(* NC axis ctrl for EL7201 via EtherCAT *)
FUNCTION_BLOCK FB_MC2_EL7201AxisCtrl
VAR_INPUT
	bEnable				: BOOL;		(* set TRUE to enable axis and drive *)
	bReset				: BOOL;		(* set TRUE to reset axis or drive from ERROR condition *)
	bEnableRevDir		: BOOL;		(* set TRUE to allow axis to run in reverse direction *)
	fOverride			: LREAL;	(* max axis output in % *)
	bFastStop			: BOOL;		(* set TRUE to override RUN signals and stop axis immediately *)
	bRunVelo			: BOOL;		(* set TRUE to run axis at specified velocity, set FALSE to stop at specified pos *)
	bStopAtPos			: BOOL;		(* set TRUE to run axis at specified velocity, set FALSE to stop at specified pos *)
	bJogFwd				: BOOL;		(* set TRUE to jog forwards *)
	bJogRev				: BOOL;		(* set TRUE to jog reverse *)
	fStopPos			: LREAL;	(* target stop position *)
	fSetVelo			: LREAL;	(* target velocity *)
	fJogVelo			: LREAL;	(* jog velocity (does not take effect if jog is in progress *)
	sRamps				: ST_AxisCtrlRamps;	(* ramps for FastStop, Normal and Jog *)
	nEtherCATState		: UINT;		(* EtherCAT operating state *)
END_VAR
VAR_IN_OUT
	sParamSet			: ST_AxisParameterSet;	(* axis parameter set *)
	sAxis				: AXIS_REF;	(* NC axis structure *)
END_VAR
VAR_OUTPUT
	bInitOK				: BOOL;		(* TRUE = parameter set read at least once *)
	bEnabled			: BOOL;		(* TRUE = axis is enabled *)
	bActive				: BOOL;		(* TRUE = axis is moving *)
	bJogActive			: BOOL;		(* TRUE = axis is moving in JOG mode *)
	bRunningFwd			: BOOL;		(* TRUE = axis is running forwards *)
	bRunningRev			: BOOL;		(* TRUE = axis is running backwards *)
	bHomed				: BOOL;		(* TRUE = axis has been homed *)
	bAxisError			: BOOL;		(* TRUE = axis is in error state *)
	nAxisErrorID		: UDINT;	(* NC axis error code *)

	fActPos				: LREAL;	(* axis absolute position *)
	fModuloPos			: LREAL;	(* axis modulo position *)
	fActVelo			: LREAL;	(* axis actual velocity *)
	bDriveError			: BOOL;		(* TRUE = EL7201 error active *)
	nStatusDWord		: DWORD;		(* drive status code *)
	fAmplifierTemp		: LREAL;	(* Amplifier temperature (degrees) *)
	fDCLinkVolts		: LREAL;	(* DC link voltage (volts) *)
END_VAR
VAR
	fbAxisCtrl			: FB_MC2_BasicAxisCtrl;
	fbEtherCATDelay		: TON;
	fbVeloCtrl			: FB_MC2_VeloCtrl;
	fbDriveReset		: MC_Reset;
	fbDriveAddr			: MC_ReadDriveAddress;
	fbDriveStatus		: FB_MC2_EL7201Status;
END_VAR
(*
-------------------------------------------------------------------------------------------------
Date		Version	Author	Comments
-------------------------------------------------------------------------------------------------
30/01/2015	3.00.00	PB		Updated with new FB_MC2_BasicAxisCtrl.
							MC_Reset for DriveReset now phased with fbSyncTimer in FB_MC2_BasicAxisCtrl.
							EL7201 status info (Warning, AmplifierTemp and DCLinkVolts) read via EtherCAT acyclic channel .
							
-------------------------------------------------------------------------------------------------
17/10/2012	1.09.02	PB		MC_Reset added to clear DriveError. as this does not cause Axis Error.
							FB_MC2_BasicAxisCtrl only issues reset if AxisError is active but DriveError on EL7201 does not cause AxisError.
21/12/2011	1.08.00	PB		Initial release

-------------------------------------------------------------------------------------------------
*)
VAR // added by the converter: edge detectors and wires of the graphical bodies
    _w1 : BOOL;
END_VAR

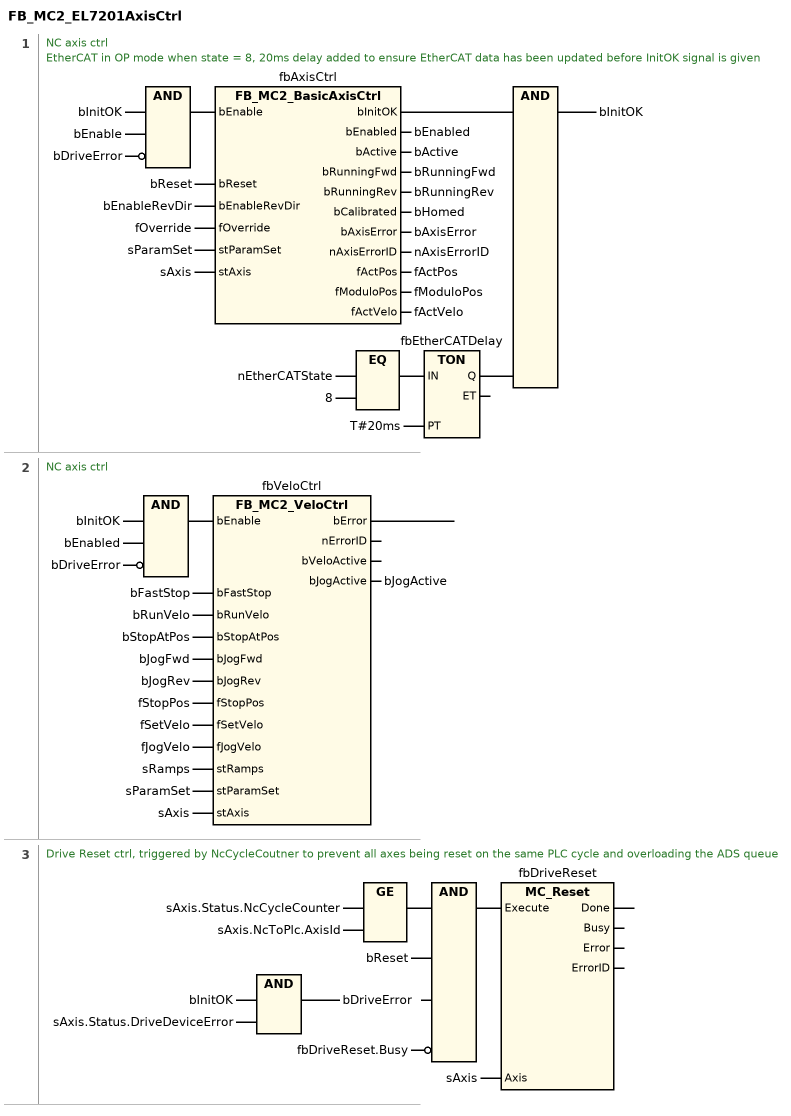
// NETWORK 1
// 					NC axis ctrl
// EtherCAT in OP mode when state = 8, 20ms delay added to ensure EtherCAT data has been updated before InitOK signal is given
//
fbAxisCtrl(
    bEnable := bInitOK AND bEnable AND NOT bDriveError,
    bReset := bReset,
    bEnableRevDir := bEnableRevDir,
    fOverride := fOverride,
    stParamSet := sParamSet,
    stAxis := sAxis,
    bEnabled => bEnabled,
    bActive => bActive,
    bRunningFwd => bRunningFwd,
    bRunningRev => bRunningRev,
    bCalibrated => bHomed,
    bAxisError => bAxisError,
    nAxisErrorID => nAxisErrorID,
    fActPos => fActPos,
    fModuloPos => fModuloPos,
    fActVelo => fActVelo); // FB_MC2_BasicAxisCtrl
fbEtherCATDelay(IN := nEtherCATState = 8, PT := T#20ms); // TON
bInitOK := fbAxisCtrl.bInitOK AND fbEtherCATDelay.Q;

// NETWORK 2
// NC axis ctrl
fbVeloCtrl(
    bEnable := bInitOK AND bEnabled AND NOT bDriveError,
    bFastStop := bFastStop,
    bRunVelo := bRunVelo,
    bStopAtPos := bStopAtPos,
    bJogFwd := bJogFwd,
    bJogRev := bJogRev,
    fStopPos := fStopPos,
    fSetVelo := fSetVelo,
    fJogVelo := fJogVelo,
    stRamps := sRamps,
    stParamSet := sParamSet,
    stAxis := sAxis,
    bJogActive => bJogActive); // FB_MC2_VeloCtrl

// NETWORK 3
// Drive Reset ctrl, triggered by NcCycleCoutner to prevent all axes being reset on the same PLC cycle and overloading the ADS queue
_w1 := bInitOK AND sAxis.Status.DriveDeviceError;
bDriveError := _w1;
fbDriveReset(Execute := sAxis.Status.NcCycleCounter >= sAxis.NcToPlc.AxisId AND bReset AND _w1 AND NOT fbDriveReset.Busy, Axis := sAxis); // MC_Reset

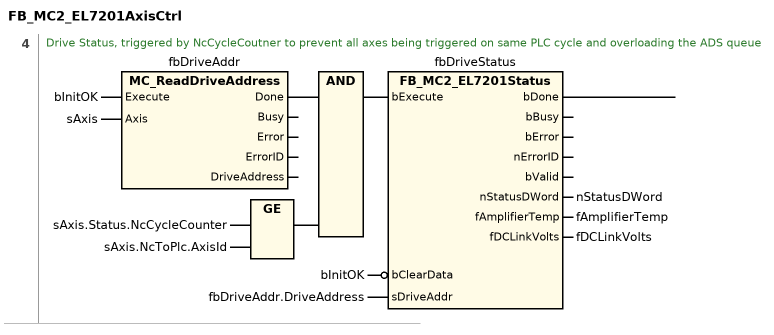
// NETWORK 4
// Drive Status, triggered by NcCycleCoutner to prevent all axes being triggered on same PLC cycle and overloading the ADS queue
fbDriveAddr(Execute := bInitOK, Axis := sAxis); // MC_ReadDriveAddress
fbDriveStatus(
    bExecute := fbDriveAddr.Done AND sAxis.Status.NcCycleCounter >= sAxis.NcToPlc.AxisId,
    bClearData := NOT bInitOK,
    sDriveAddr := fbDriveAddr.DriveAddress,
    nStatusDWord => nStatusDWord,
    fAmplifierTemp => fAmplifierTemp,
    fDCLinkVolts => fDCLinkVolts); // FB_MC2_EL7201Status

END_FUNCTION_BLOCK

(* stored: Version 1.1.0.1, ProductVersion 3.1.4024.15
   POU FB_MC2_EL7201AxisCtrl: Id {77169ede-ff04-4100-a904-5d143cc92112}, SpecialFunc None *)
